DATA_BLOCK "DB_LUZ_Type"
TITLE =%version: 0.14 % CN: 20
//History:
//This version  %created_by:   nlhdl %
//              %date_created:   Wednesday, November 01, 2017 9:02:33 AM %
//              %release: VI_RAW/RA_Dev %
//
//Modification History:                                   By:    Date:     Rev:
//----------------------------------------------------  -------  --------  -----
//ra#24938: Wrong family for multiple RAW blocks        nlHdL    01-11-17   0.14
//ra#51111:Code Update                                  inajos   29-03-17   0.13
//ra#50810: Align as per PB and Area HMI                inajos   21-03-17   0.12
//ra#18174: DI NON_RETAIN PLC Memory                    nlHdL    14-12-16   0.11
//ra#18629: Add LSZ and LUZ to the RAW Library          nlHdL    17-11-16   0.10
//ra#18629: Add LSZ and LUZ to the RAW Library          nlHdL    17-11-16   0.10
//7324: ECS-P General from the RD to RA for platform    nlHdL    06-07-15   0.10
//15797: Keyword release added                          nlwwij   26-09-13   0.10
//PR14608 Fixed mode Overal/General status changed      nlple    17-09-13   0.09
//PR9463 Add status direction not allowed               nlple    26-03-13   0.08
//PR9463 PEC gap switch added                           nlple    20-03-13   0.07
//CR8764 Changing name LUZ01 to LUZ                     nlple    13-03-12   0.06
//CR8366 Add spare bit Spare_0_4 + minor update         nlple    16-12-11   0.05
//CR6232 OP state Up/Down not reported to OP            nlple    10-01-11   0.04
//Updated to Coding conventions                         nlJBax   23-09-10   0.03
//CR5188 Updated to Coding conventions                  nlHdL    16-09-10   0.02
//Initial revision                                      insmahi  18-08-10   0.01
//
FAMILY : RAW
VERSION : 0.0
NON_RETAIN


  STRUCT
   Type_Component : BYTE ;	//Type of the component (1 = Section, 0 = Other)
   Record_Length : BYTE ;	//Number of the Detailed Status in the UDT
   Status : ARRAY  [1 .. 16 ] OF "UDT_Comp_Status";
  END_STRUCT ;
BEGIN
   Type_Component := B#16#0;
   Record_Length := B#16#16;
   Status[1].HMI_Text_Number := -1;
   Status[1].Overall_Status_Relation := B#16#5;
   Status[1].General_Status_Relation := B#16#4;
   Status[2].HMI_Text_Number := -1;
   Status[2].Overall_Status_Relation := B#16#5;
   Status[2].General_Status_Relation := B#16#4;
   Status[3].HMI_Text_Number := -1;
   Status[3].Overall_Status_Relation := B#16#0;
   Status[3].General_Status_Relation := B#16#0;
   Status[4].HMI_Text_Number := -1;
   Status[4].Overall_Status_Relation := B#16#0;
   Status[4].General_Status_Relation := B#16#0;
   Status[5].HMI_Text_Number := -1;
   Status[5].Overall_Status_Relation := B#16#0;
   Status[5].General_Status_Relation := B#16#0;
   Status[6].HMI_Text_Number := -1;
   Status[6].Overall_Status_Relation := B#16#0;
   Status[6].General_Status_Relation := B#16#0;
   Status[7].HMI_Text_Number := -1;
   Status[7].Overall_Status_Relation := B#16#0;
   Status[7].General_Status_Relation := B#16#0;
   Status[8].HMI_Text_Number := -1;
   Status[8].Overall_Status_Relation := B#16#0;
   Status[8].General_Status_Relation := B#16#0;
   Status[9].HMI_Text_Number := 352;
   Status[9].Overall_Status_Relation := B#16#4;
   Status[9].General_Status_Relation := B#16#3;
   Status[10].HMI_Text_Number := 353;
   Status[10].Overall_Status_Relation := B#16#5;
   Status[10].General_Status_Relation := B#16#4;
   Status[11].HMI_Text_Number := -1;
   Status[11].Overall_Status_Relation := B#16#0;
   Status[11].General_Status_Relation := B#16#0;
   Status[12].HMI_Text_Number := -1;
   Status[12].Overall_Status_Relation := B#16#0;
   Status[12].General_Status_Relation := B#16#0;
   Status[13].HMI_Text_Number := -1;
   Status[13].Overall_Status_Relation := B#16#0;
   Status[13].General_Status_Relation := B#16#0;
   Status[14].HMI_Text_Number := -1;
   Status[14].Overall_Status_Relation := B#16#0;
   Status[14].General_Status_Relation := B#16#0;
   Status[15].HMI_Text_Number := -1;
   Status[15].Overall_Status_Relation := B#16#0;
   Status[15].General_Status_Relation := B#16#0;
   Status[16].HMI_Text_Number := -1;
   Status[16].Overall_Status_Relation := B#16#0;
   Status[16].General_Status_Relation := B#16#0;
END_DATA_BLOCK

